TYPE ST_DetectDiameterCommand EXTENDS ST_CommandBasic :
STRUCT
	GetPhotoCompleted : BOOL;
END_STRUCT
END_TYPE

(* stored: Version 1.1.0.1, ProductVersion 3.1.4024.13
   DUT ST_DetectDiameterCommand: Id {3ddfdeb5-5f6a-4df6-a8b4-452e39e5bfb3} *)
